// TIA Portal V16 export
// export: Created 2024-12-03T15:41:44.8807353Z, ExportSetting WithReadOnly, DisplayName Totally Integrated Automation Portal, DisplayVersion V16 Update 6, DisplayName TIA Portal Version Control Interface, DisplayVersion V16 Update 2, DisplayName TIA Portal Openness, DisplayVersion V16 Update 6, DisplayName TIA Portal Teamcenter Gateway, DisplayVersion V16, DisplayName SINAMICS Startdrive Advanced, DisplayVersion V16 Update 5, DisplayName SINAMICS Startdrive G130, G150, S120, S150, SINAMICS MV, S210, DisplayVersion V16 Update 5, DisplayName SINAMICS Startdrive G110M, G120, G120C, G120D, G120P, G115D, DisplayVersion V16 Update 5, DisplayName STEP 7 Professional, DisplayVersion V16 Update 6, DisplayName STEP 7 Safety, DisplayVersion V16, DisplayName WinCC Advanced / Unified PC, DisplayVersion V16 Update 6
TYPE "Cylinder_UDT"
// stored: CreationDate 2021-10-04T17:07:47.657452Z, InterfaceModifiedDate 2021-10-04T17:08:20.2971293Z, IsConsistent true, LibraryConformanceStatus The object is library-conformant., ModifiedDate 2021-10-04T17:08:20.2971293Z
   STRUCT
      Cmd : Struct
         InAuto : Bool;
         OutAuto : Bool;
         InManual : Bool;
         OutManual : Bool;
         InManualHMI : Bool;
         OutManualHMI : Bool;
         Interlock : Bool;
      END_STRUCT;
      Alarms : Struct
         NotIn : "HmiAlarm";   // Object in feedback not received in time
         NotOut : "HmiAlarm";   // Object out feedback not received in time
         Status : Word;   // lsb 0 not in | lsb 1 not out
      END_STRUCT;
      Status : Struct
         Position : Int;   // 0 Traveling | 1 out | -1 in
         ManualModeActive : Bool;
         ManualCommandsDisabled : Bool;
         Interlocked : Bool;
         status : Word;   // lsb 0 Interlocked | lsb 1 manual mode active
      END_STRUCT;
      Settings : Struct
         feedBackInDelay : Time;
         feedBackOutDelay : Time;
         CylinderInTime : Time := t#5s;
         CylinderOutTime : Time := t#5s;
         CmdOnError : Bool;   // Copy all the commends when leaving manual mode or auto mode
         CopyCommands : Bool;
         CylinderType : Int;   // (0 bistabiel) (1 monostabiel rest in) (2 monostabiel rest out)
         EnableManualIn : Bool := true;
         EnableManualOut : Bool := true;
      END_STRUCT;
      "Name" : String[40];
      Zone : Int;
   END_STRUCT;
END_TYPE
